FUNCTION_BLOCK AsyncResponseSessionData_TestSuite EXTENDS TcUnit.FB_TestSuite
VAR
END_VAR

TestNewResponseIsPending();
TestFreshResponseHasNotExpired();
TestZeroMaxAgeDisablesTheDeadline();
TestCompletedResponseIsNoLongerPending();
TestRejectedResponseIsNoLongerPending();

METHOD TestCompletedResponseIsNoLongerPending
VAR
	asyncResponseSessionData : AsyncResponseSessionData(SuggestedRetryDelayInMs := 0, MaxAge := T#60S);
END_VAR
TEST('TestCompletedResponseIsNoLongerPending');

asyncResponseSessionData.Success();

AssertFalse(
	Condition := asyncResponseSessionData.IsPending,
	Message := 'A response which has completed should no longer report as pending'
);

TEST_FINISHED();
END_METHOD

METHOD TestFreshResponseHasNotExpired
VAR
	asyncResponseSessionData : AsyncResponseSessionData(SuggestedRetryDelayInMs := 0, MaxAge := T#60S);
END_VAR
TEST('TestFreshResponseHasNotExpired');

AssertFalse(
	Condition := asyncResponseSessionData.HasExpired,
	Message := 'A response created this cycle cannot already be past a 60s deadline'
);

TEST_FINISHED();
END_METHOD

METHOD TestNewResponseIsPending
VAR
	asyncResponseSessionData : AsyncResponseSessionData(SuggestedRetryDelayInMs := 0, MaxAge := T#60S);
END_VAR
TEST('TestNewResponseIsPending');

AssertTrue(
	Condition := asyncResponseSessionData.IsPending,
	Message := 'A newly created response should be pending until the handler completes it'
);

TEST_FINISHED();
END_METHOD

METHOD TestRejectedResponseIsNoLongerPending
VAR
	asyncResponseSessionData : AsyncResponseSessionData(SuggestedRetryDelayInMs := 0, MaxAge := T#60S);
END_VAR
TEST('TestRejectedResponseIsNoLongerPending');

asyncResponseSessionData.Error('SOME_CODE', 'some message');

AssertFalse(
	Condition := asyncResponseSessionData.IsPending,
	Message := 'A response which has been rejected should no longer report as pending'
);

TEST_FINISHED();
END_METHOD

METHOD TestZeroMaxAgeDisablesTheDeadline
VAR
	asyncResponseSessionData : AsyncResponseSessionData(SuggestedRetryDelayInMs := 0, MaxAge := T#0S);
END_VAR
TEST('TestZeroMaxAgeDisablesTheDeadline');

// T#0S is the documented way to switch the deadline off.  It must not be read
// as 'expires immediately', which would fail every asynchronous call.
AssertFalse(
	Condition := asyncResponseSessionData.HasExpired,
	Message := 'A max age of T#0S should disable the deadline, not expire instantly'
);

TEST_FINISHED();
END_METHOD

END_FUNCTION_BLOCK

(* stored: Version 1.1.0.1, ProductVersion 3.1.4026.13
   POU AsyncResponseSessionData_TestSuite: Id {7b3d5c81-40e9-0a72-6c15-93f2ad81be40}, SpecialFunc None
   Method TestCompletedResponseIsNoLongerPending: Id {2c8f14a6-9b03-05de-4471-8e6a2f0517cb}
   Method TestFreshResponseHasNotExpired: Id {5a190b73-6e24-0c38-1f07-b6d4029ae5f1}
   Method TestNewResponseIsPending: Id {9d0e2f47-1c85-0b16-3a92-47f18c60d3ea}
   Method TestRejectedResponseIsNoLongerPending: Id {4f62b0d9-83a1-0e57-25cb-1a09df73b268}
   Method TestZeroMaxAgeDisablesTheDeadline: Id {8e15c3a2-27b6-0f49-59d3-c0b842e19a75} *)
